// Mitsubishi GX Works2 project: group_26_PLC _Noam   PLC: FX3G

// global labels: Global1
VAR_GLOBAL
  start_work_day AT X007 : BOOL;
  lamp_y7 AT Y007 : BOOL;
  end_day AT M7 : BOOL;
  lamp_work_day AT Y007 : BOOL;
  emrgency AT X005 : BOOL;
  chocolate_stock AT D1100 : REAL;
  nuts_stock AT D1102 : REAL;
  pistachio_stock AT D1105 : REAL;
  kadaif_stock AT D1107 : REAL;
  melting_process AT X001 : BOOL;
END_VAR
VAR_GLOBAL CONSTANT
  ch : REAL := 300;
  const_400 : REAL := 400;
END_VAR
VAR_GLOBAL
  melting_stock AT D1109 : REAL;
  melting_lamp AT Y001 : BOOL;
  temp_45 AT X002 : BOOL;
  finish_transfer AT M1 : BOOL;
  finish_melting AT M2 : BOOL;
  empty_templates AT X003 : BOOL;
  casting_stock AT D1111 : REAL;
END_VAR
VAR_GLOBAL CONSTANT
  const50 : INT := 50;
END_VAR
VAR_GLOBAL
  casting_process AT Y002 : BOOL;
  casting_timer AT TC1 : BOOL;
  casting_timer_on AT TS1 : BOOL;
  filing AT X004 : BOOL;
  analog_input1 AT D8280 : INT;
  log_input AT D1111 : INT;
  normal_input AT D1200 : REAL;
END_VAR
VAR_GLOBAL CONSTANT
  const_5 : REAL := 5;
END_VAR
VAR_GLOBAL
  nuts AT M4 : BOOL;
  dubai AT M5 : BOOL;
END_VAR
VAR_GLOBAL CONSTANT
  const_100 : REAL := 100;
END_VAR
VAR_GLOBAL
  fill_nuts AT D1113 : REAL;
  filling_stock AT D1113 : REAL;
END_VAR
VAR_GLOBAL CONSTANT
  const_20 : REAL := 20;
  const_120 : REAL := 120;
  const_60 : REAL := 60;
END_VAR
VAR_GLOBAL
  save_analog AT D1250 : REAL;
  save_analog1 AT D1250 : REAL;
  real_input AT D1200 : REAL;
END_VAR
VAR_GLOBAL CONSTANT
  const_6 : REAL := 6;
END_VAR
VAR_GLOBAL
  filling_cream AT M6 : BOOL;
  filling_timer AT TC2 : BOOL;
END_VAR
VAR_GLOBAL CONSTANT
  const40 : INT := 40;
  const_50 : INT := 50;
  const5 : INT := 5;
END_VAR
VAR_GLOBAL
  flicker3_on AT TS3 : BOOL;
  lamp3 AT Y003 : BOOL;
  flicker4 AT TC4 : BOOL;
  flicker4_on AT TS4 : BOOL;
  lamp4 AT Y004 : BOOL;
  flicker AT M8 : BOOL;
  flickerr3 AT TC3 : BOOL;
  filling_timer_on1 AT TS2 : BOOL;
  cooling AT X006 : BOOL;
END_VAR
VAR_GLOBAL CONSTANT
  const_30 : INT := 30;
END_VAR
VAR_GLOBAL
  cooling_timer AT TS5 : BOOL;
  cooling_time AT M9 : BOOL;
  cooling_process AT Y006 : BOOL;
END_VAR
VAR_GLOBAL CONSTANT
  const_40 : INT := 40;
END_VAR
VAR_GLOBAL
  pack1 AT X000 : BOOL;
  finish_pack AT M10 : BOOL;
  count_chocolate AT CS0 : BOOL;
END_VAR
VAR_GLOBAL CONSTANT
  count1 : REAL := 1;
END_VAR
VAR_GLOBAL
  count_to_4 AT CC1 : BOOL;
END_VAR
VAR_GLOBAL CONSTANT
  count4 : INT := 4;
END_VAR
VAR_GLOBAL
  count_first AT CS0 : BOOL;
  count_last AT CS1 : BOOL;
  packing_light AT Y005 : BOOL;
  cooling_timer_tc AT TC5 : BOOL;
  conut_last_help AT M11 : BOOL;
END_VAR
VAR_GLOBAL CONSTANT
  const40packeges : REAL := 40.0;
END_VAR
VAR_GLOBAL
  output_packs AT D8282 : INT;
END_VAR
VAR_GLOBAL CONSTANT
  const_0 : REAL;
END_VAR
VAR_GLOBAL
  analog_pack AT D1252 : REAL;
  all_packeges AT D1117 : REAL;
  input_chocolate AT D1120 : REAL;
  input_nuts AT D1122 : REAL;
  input_pistachio AT D1124 : REAL;
  input_kadaif AT D1126 : REAL;
  no_inventory AT M14 : BOOL;
END_VAR
VAR_GLOBAL CONSTANT
  amount_nuts_for_mix : REAL := 100;
  amount_pistachio_for_mix : REAL := 120;
END_VAR
VAR_GLOBAL
  valid_stock_mix AT M15 : BOOL;
  valid_stock_dubai AT M16 : BOOL;
END_VAR
VAR_GLOBAL CONSTANT
  amount_kadaif : REAL := 60;
  amount_pistachio : REAL := 120;
  amount_nuts : REAL := 100;
  amount_chocolate : REAL := 400;
END_VAR
VAR_GLOBAL
  nuts_pick AT M21 : BOOL;
  help_input AT X010 : BOOL;
END_VAR

// task Task_01 (event TRUE, interval 0, priority 31): POU_01

PROGRAM POU_01
VAR
  casting_time : BOOL;
  filling_timer_on : BOOL;
  flicker3 : BOOL;
END_VAR
(* structured ladder/FBD written out as ST: instructions are called as NAME(EN, inputs, outputs); _pN, _eN, _tN stand for wires *)
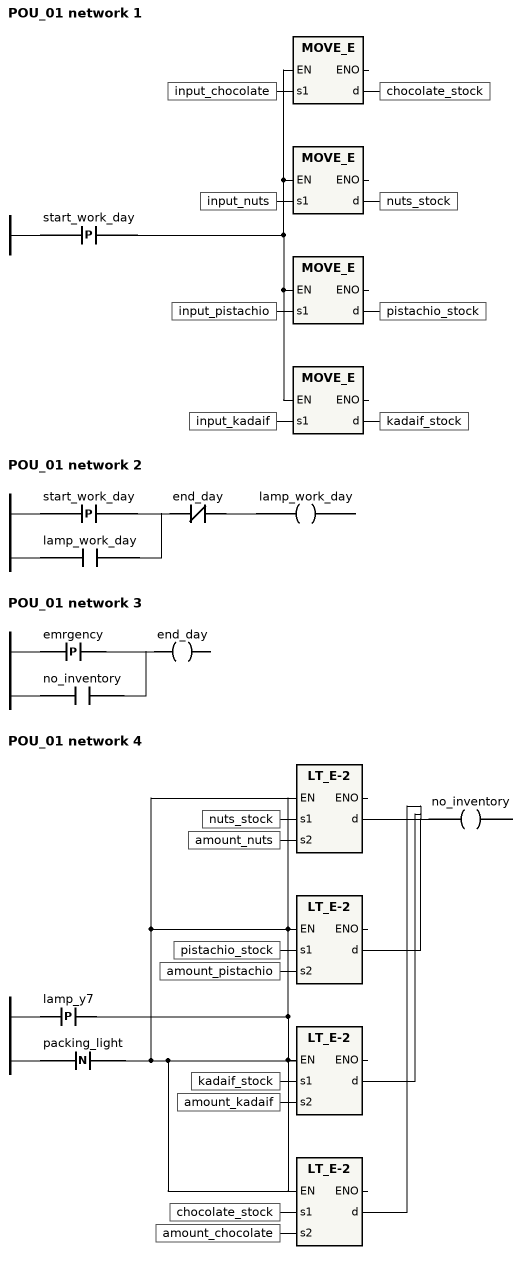
(* network 1 *)
_p1 := LDP(TRUE, start_work_day);
MOVE_E(_p1, input_chocolate, chocolate_stock);
MOVE_E(_p1, input_nuts, nuts_stock);
MOVE_E(_p1, input_pistachio, pistachio_stock);
MOVE_E(_p1, input_kadaif, kadaif_stock);
(* network 2 *)
lamp_work_day := (LDP(TRUE, start_work_day) OR lamp_work_day) AND NOT end_day;
(* network 3 *)
end_day := LDP(TRUE, emrgency) OR no_inventory;
(* network 4 *)
_p1 := LDP(TRUE, lamp_y7) OR LDF(TRUE, packing_light);
LT_E(_p1, nuts_stock, amount_nuts, _t2);
LT_E(_p1, pistachio_stock, amount_pistachio, _t3);
LT_E(_p1, kadaif_stock, amount_kadaif, _t4);
LT_E(_p1, chocolate_stock, amount_chocolate, _t5);
no_inventory := _t2 OR _t3 OR _t4 OR _t5;
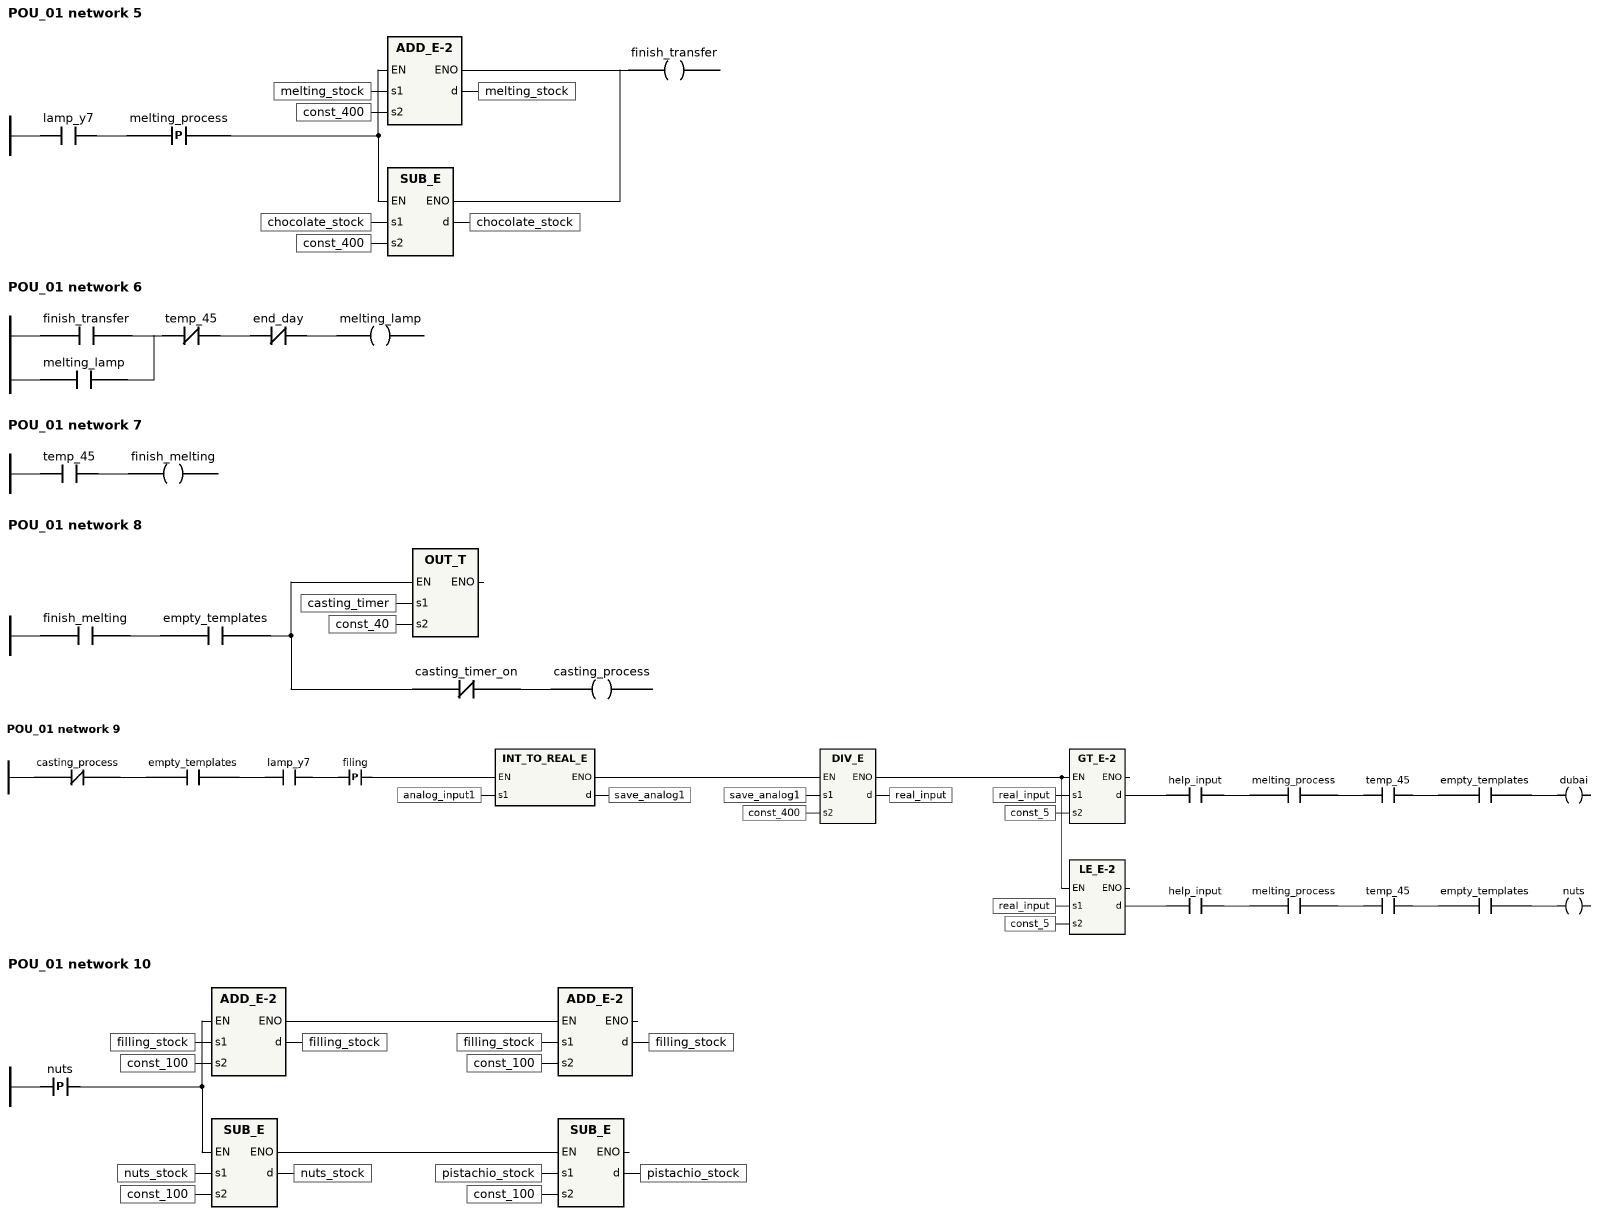
(* network 5 *)
_p1 := lamp_y7 AND LDP(TRUE, melting_process);
_e2 := ADD_E(_p1, melting_stock, const_400, melting_stock);
_e3 := SUB_E(_p1, chocolate_stock, const_400, chocolate_stock);
finish_transfer := _e2 OR _e3;
(* network 6 *)
melting_lamp := ((finish_transfer OR melting_lamp) AND NOT temp_45) AND NOT end_day;
(* network 7 *)
finish_melting := temp_45;
(* network 8 *)
_p1 := finish_melting AND empty_templates;
OUT_T(_p1, casting_timer, const_40);
casting_process := _p1 AND NOT casting_timer_on;
(* network 9 *)
_e1 := INT_TO_REAL_E(NOT casting_process AND empty_templates AND lamp_y7 AND LDP(TRUE, filing), analog_input1, save_analog1);
_e2 := DIV_E(_e1, save_analog1, const_400, real_input);
GT_E(_e2, real_input, const_5, _t3);
dubai := _t3 AND help_input AND melting_process AND temp_45 AND empty_templates;
LE_E(_e2, real_input, const_5, _t4);
nuts := _t4 AND help_input AND melting_process AND temp_45 AND empty_templates;
(* network 10 *)
_p1 := LDP(TRUE, nuts);
_e2 := ADD_E(_p1, filling_stock, const_100, filling_stock);
ADD_E(_e2, filling_stock, const_100, filling_stock);
_e3 := SUB_E(_p1, nuts_stock, const_100, nuts_stock);
SUB_E(_e3, pistachio_stock, const_100, pistachio_stock);
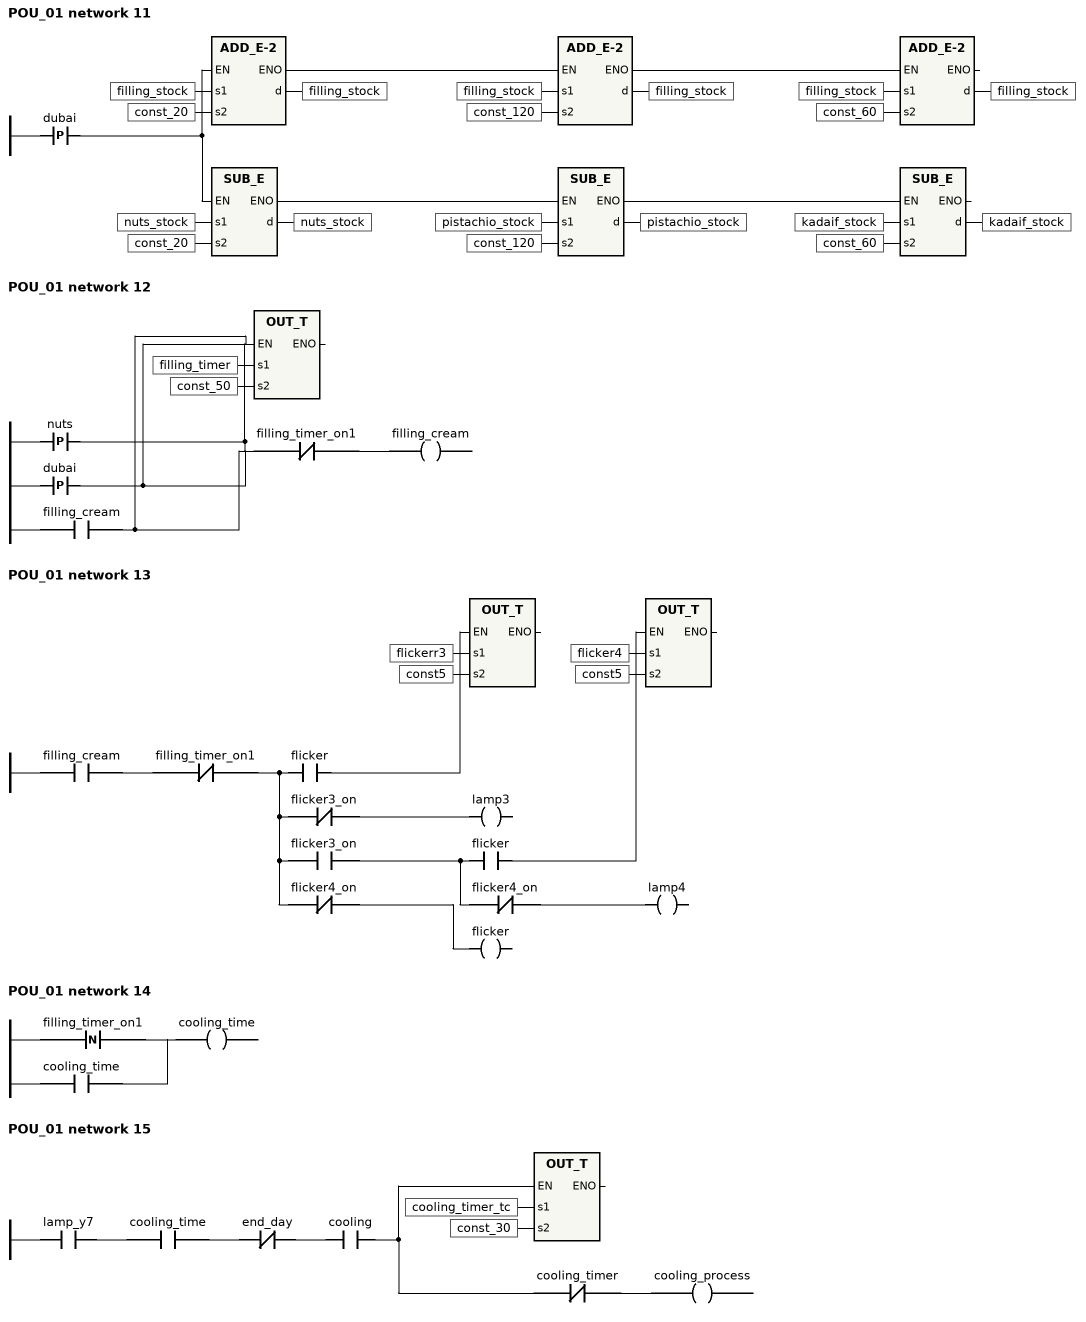
(* network 11 *)
_p1 := LDP(TRUE, dubai);
_e2 := ADD_E(_p1, filling_stock, const_20, filling_stock);
_e3 := ADD_E(_e2, filling_stock, const_120, filling_stock);
ADD_E(_e3, filling_stock, const_60, filling_stock);
_e4 := SUB_E(_p1, nuts_stock, const_20, nuts_stock);
_e5 := SUB_E(_e4, pistachio_stock, const_120, pistachio_stock);
SUB_E(_e5, kadaif_stock, const_60, kadaif_stock);
(* network 12 *)
_p1 := LDP(TRUE, nuts) OR LDP(TRUE, dubai) OR filling_cream;
OUT_T(_p1, filling_timer, const_50);
filling_cream := _p1 AND NOT filling_timer_on1;
(* network 13 *)
_p1 := filling_cream AND NOT filling_timer_on1;
OUT_T(_p1 AND flicker, flickerr3, const5);
lamp3 := _p1 AND NOT flicker3_on;
_p2 := _p1 AND flicker3_on;
OUT_T(_p2 AND flicker, flicker4, const5);
lamp4 := _p2 AND NOT flicker4_on;
flicker := _p1 AND NOT flicker4_on;
(* network 14 *)
cooling_time := LDF(TRUE, filling_timer_on1) OR cooling_time;
(* network 15 *)
_p1 := lamp_y7 AND cooling_time AND NOT end_day AND cooling;
OUT_T(_p1, cooling_timer_tc, const_30);
cooling_process := _p1 AND NOT cooling_timer;
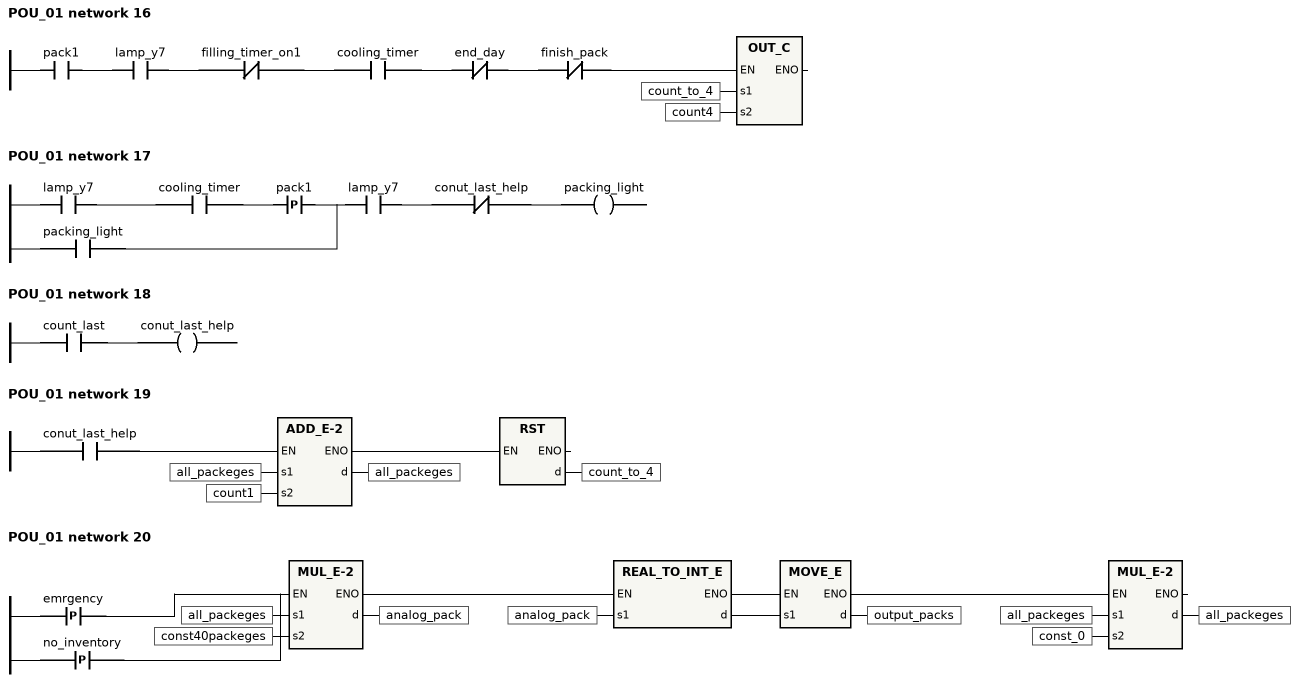
(* network 16 *)
OUT_C(pack1 AND lamp_y7 AND NOT filling_timer_on1 AND cooling_timer AND NOT end_day AND NOT finish_pack, count_to_4, count4);
(* network 17 *)
packing_light := (((lamp_y7 AND cooling_timer AND LDP(TRUE, pack1)) OR packing_light) AND lamp_y7) AND NOT conut_last_help;
(* network 18 *)
conut_last_help := count_last;
(* network 19 *)
_e1 := ADD_E(conut_last_help, all_packeges, count1, all_packeges);
RST(_e1, count_to_4);
(* network 20 *)
_e1 := MUL_E(LDP(TRUE, emrgency) OR LDP(TRUE, no_inventory), all_packeges, const40packeges, analog_pack);
_e3 := REAL_TO_INT_E(_e1, analog_pack, _t2);
_e4 := MOVE_E(_e3, _t2, output_packs);
MUL_E(_e4, all_packeges, const_0, all_packeges);
END_PROGRAM
